FUNCTION_BLOCK EL2732
VAR
	{attribute addProperty Name "WcState"}
	_wcState : WcStateBase;
	{attribute addProperty Name "Info data"}
	_infoData : InfoDataBase;
	_io : EL2xx2_Data;
END_VAR

PROPERTY IO : REFERENCE TO EL2xx2_Data
GET
IO REF= _io;
END_GET
END_PROPERTY

PROPERTY WcState : REFERENCE TO WcStateBase
GET
WcState REF= _wcState;
END_GET
END_PROPERTY

END_FUNCTION_BLOCK

(* stored: Version 1.1.0.1, ProductVersion 3.1.4024.9
   POU EL2732: Id {0c52c089-e53a-0ccb-36fd-77cf3b8a8e9a}, SpecialFunc None
   Property IO: Id {90744fd5-be8c-0563-3270-1c181ae81943}
   Get Get: Id {aa07a8a7-18f0-02a8-1647-9e8c598c929b}
   Property WcState: Id {4e087e6a-fee1-085b-032a-8a8b28ddf23d}
   Get Get: Id {3c9c4730-3e92-032a-1b94-60a701fbc938} *)
